// TIA Portal V21 export
TYPE "LAxisCtrl_typeGearInAbsolute"
TITLE = LAxisCtrl_typeGearInAbsolute
// Support: tech.team.motioncontrol@siemens.com
   STRUCT
      ratioNumerator : DInt := 1;   // Gear ratio numerator (permitted integer values: -2147483648 to 2147483647; value 0 not permitted)
      ratioDenominator : DInt := 1;   // Gear ratio denominator (permitted integer values: 1 to 2147483647)
      masterSyncPosition : LReal := 0.0;   // Synchronous position of leading axis
      slaveSyncPosition : LReal := 0.0;   // Synchronous position of following axis
      syncProfileReference : DInt := 1;   // Type of synchronization (0: Synchronization in advance using dynamic parameters; 1: Synchronization in advance using leading value distance; 3: Subsequent synchronization using leading value distance)
      masterStartDistance : LReal := 0.0;   // Leading value distance when "SyncProfileReference" = 1, 3
      velocity : LReal := -1.0;   // Velocity for synchronization (Value > 0.0: The specified value is used; Value = 0.0: Not permitted; Value < 0.0: Use of the default value configured in the technology object) when "SyncProfileReference" = 0
      acceleration : LReal := -1.0;   // Acceleration for synchronization (Value > 0.0: The specified value is used; Value = 0.0: Not permitted; Value < 0.0: Use of the default value configured in the technology object) when "SyncProfileReference" = 0
      deceleration : LReal := -1.0;   // Deceleration for synchronization (Value > 0.0: The specified value is used; Value = 0.0: Not permitted; Value < 0.0: Use of the default value configured in the technology object) when "SyncProfileReference" = 0
      jerk : LReal := -1.0;   // Jerk for synchronization (Value > 0.0: Smooth velocity profile, the specified value is used; Value = 0.0: Trapezoid velocity profile; Value < 0.0: Use of the default value configured in the technology object) when "SyncProfileReference" = 0
      syncDirection : DInt := 1;   // Direction for synchronization only in effect for axes with activated modulo setting (1: Forward direction; 2: Backward direction; 3: Shortest way)
      ratioChangeOnTheFly : Bool := FALSE;   // TRUE: Changing gear ratio on-the-fly; FALSE: Ratio change requires a new rising edge at gearInAbsolute input
   END_STRUCT;
END_TYPE
